(* IEC 61131-3 sources: CodesysTest/export/Unused/FB_SimBasicBagDelivery.pou/BagFeedDone.prop, 1 file *)

(* ---- Get.pm.st ---- *)
(*#-#-#-#-#-#-#-#-#-#---Declaration---#-#-#-#-#-#-#-#-#-#-#-#-#*)

VAR
END_VAR
(*#-#-#-#-#-#-#-#-#-#---Implementation---#-#-#-#-#-#-#-#-#-#-#-#-#*)

BagFeedDone := feedBagOut.Q;
